(* Logix 5000 project; controller GP1 vendor 1 type 14 code 155 rev 32.11; software revision 32.01; part 2 of 2 *)
(* tags used below, declared in another part *)
   CERRARSESION : BOOL;
   ING_ACCESS : BOOL;
   LOGOUT : BOOL;
   MTTO_ACCESS : BOOL;
   ACT1_OFF : BOOL;   // TROQUEL OFF
   ACT2_OFF : BOOL;   // CORTE SUPERIOR OFF
   ACT3_OFF : BOOL;   // NAVAJA 1 OFF
   ACT5_OFF : BOOL;   // CLAMP OFF
   EVBI0_AUTO_OFF : BOOL;   // NAVAJAS 3 OFF AUTO
   EVBI0_AUTO_ON : BOOL;   // NAVAJAS 3 ON AUTO
   EVBI0_MAN_OFF : BOOL;   // NAVAJAS 3 OFF MANUAL
   EVBI0_MAN_ON : BOOL;   // NAVAJAS 3 ON MANUAL
   EVBI0_OFF : BOOL;   // NAVAJAS 3 OFF
   EVBI0_ON : BOOL;   // NAVAJAS 3 ON
   EVBI1_AUTO_OFF : BOOL;   // TROQUEL OFF AUTO
   EVBI1_AUTO_ON : BOOL;   // TROQUEL ON AUTO
   EVBI1_MAN_OFF : BOOL;   // TROQUEL OFF MANUAL
   EVBI1_MAN_ON : BOOL;   // TROQUEL ON MANUAL
   EVBI1_OFF : BOOL;   // TROQUEL OFF
   EVBI1_ON : BOOL;   // TROQUEL ON
   EVBI2_AUTO_OFF : BOOL;   // CLAMP OFF AUTO
   EVBI2_AUTO_ON : BOOL;   // CLAMP ON AUTO
   EVBI2_MAN_OFF : BOOL;   // CLAMP OFF MANUAL
   EVBI2_MAN_ON : BOOL;   // CLAMP ON MANUAL
   EVBI2_OFF : BOOL;   // CLAMP OFF
   EVBI2_ON : BOOL;   // CLAMP ON
   EVBI3_AUTO_OFF : BOOL;   // NAVAJA 1 OFF AUTO
   EVBI3_AUTO_ON : BOOL;   // NAVAJA 1 ON AUTO
   EVBI3_MAN_OFF : BOOL;   // NAVAJA 1 OFF MANUAL
   EVBI3_MAN_ON : BOOL;   // NAVAJA 1 ON MANUAL
   EVBI3_OFF : BOOL;   // NAVAJA 1 OFF
   EVBI3_ON : BOOL;   // NAVAJA 1 ON
   EVBI4_OFF : BOOL;   // CLAMP VERTICAL OFF
   EVBI4_ON : BOOL;   // CLAMP VERTICAL ON
   EVBI5_AUTO_OFF : BOOL;   // CORTE SUPERIOR OFF AUTO
   EVBI5_AUTO_ON : BOOL;   // CORTE SUPERIOR ON AUTO
   EVBI5_MAN_OFF : BOOL;   // CORTE SUPERIOR OFF MANUAL
   EVBI5_MAN_ON : BOOL;   // CORTE SUPERIOR ON MANUAL
   EVBI5_OFF : BOOL;   // CORTE SUPERIOR OFF
   EVBI5_ON : BOOL;   // CORTE SUPERIOR ON
   EVBI6_OFF : BOOL;   // CLAMP HORIZONTAL OFF
   EVBI6_ON : BOOL;   // CLAMP HORIZONTAL ON
   EVMONO1_AUTO_ON : BOOL;   // TOPE_AUTO_ON
   EVMONO1_MAN_ON : BOOL;
   EVMONO_ON : BOOL;   // TOPE ON
   REARMY_BUTTON : BOOL;
   RESET_COUNTER : BOOL;
   TCLAMP : TIMER;
   USER : DINT;
   WORKING : BOOL;
(* MainProgram, continued *)

ROUTINE OUTPUTS   (* ladder *)
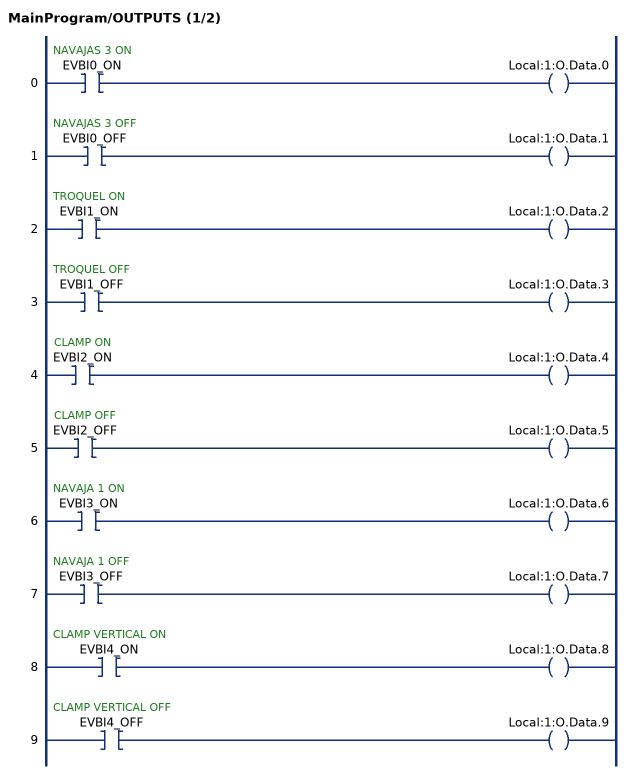
   0: XIC(EVBI0_ON)OTE(Local:1:O.Data.0);
   1: XIC(EVBI0_OFF)OTE(Local:1:O.Data.1);
   2: XIC(EVBI1_ON)OTE(Local:1:O.Data.2);
   3: XIC(EVBI1_OFF)OTE(Local:1:O.Data.3);
   4: XIC(EVBI2_ON)OTE(Local:1:O.Data.4);
   5: XIC(EVBI2_OFF)OTE(Local:1:O.Data.5);
   6: XIC(EVBI3_ON)OTE(Local:1:O.Data.6);
   7: XIC(EVBI3_OFF)OTE(Local:1:O.Data.7);
   8: XIC(EVBI4_ON)OTE(Local:1:O.Data.8);
   9: XIC(EVBI4_OFF)OTE(Local:1:O.Data.9);
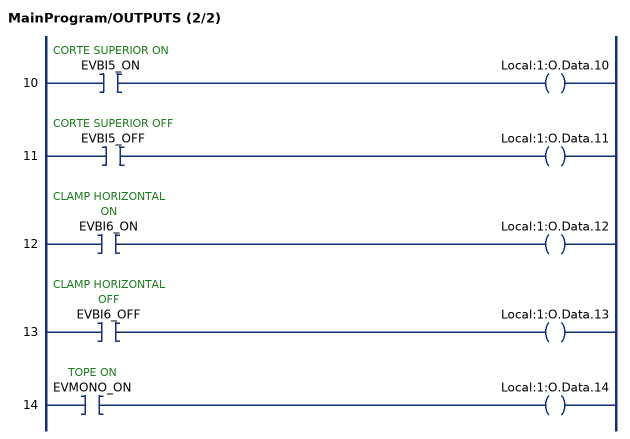
   10: XIC(EVBI5_ON)OTE(Local:1:O.Data.10);
   11: XIC(EVBI5_OFF)OTE(Local:1:O.Data.11);
   12: XIC(EVBI6_ON)OTE(Local:1:O.Data.12);
   13: XIC(EVBI6_OFF)OTE(Local:1:O.Data.13);
   14: XIC(EVMONO_ON)OTE(Local:1:O.Data.14);
END_ROUTINE

ROUTINE USERS   (* ladder *)
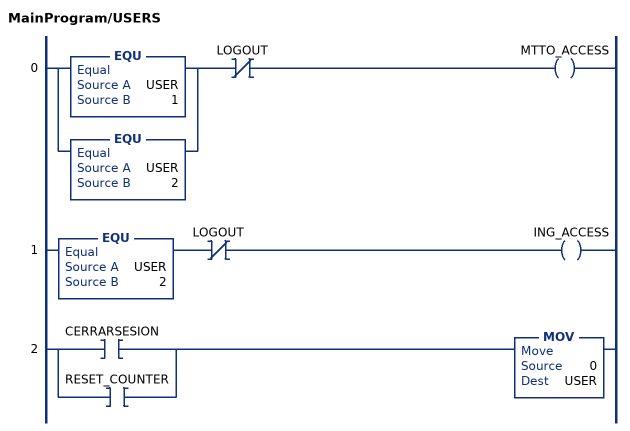
   0: [EQU(USER,1) ,EQU(USER,2) ]XIO(LOGOUT)OTE(MTTO_ACCESS);
   1: EQU(USER,2)XIO(LOGOUT)OTE(ING_ACCESS);
   2: [XIC(CERRARSESION) ,XIC(RESET_COUNTER) ]MOV(0,USER);
END_ROUTINE

ROUTINE VALVES_ACTIV   (* ladder *)
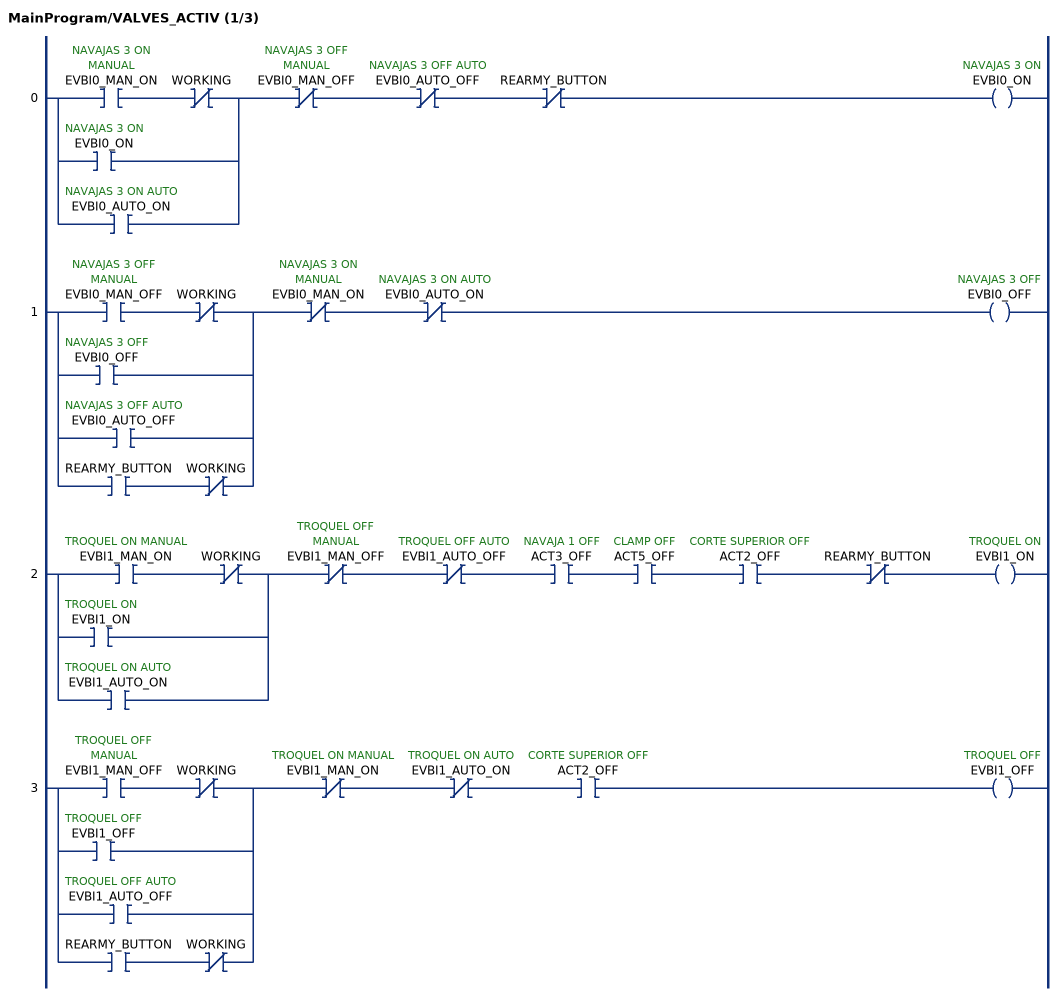
   0: [XIC(EVBI0_MAN_ON) XIO(WORKING) ,XIC(EVBI0_ON) ,XIC(EVBI0_AUTO_ON) ]XIO(EVBI0_MAN_OFF)XIO(EVBI0_AUTO_OFF)XIO(REARMY_BUTTON)OTE(EVBI0_ON);
   1: [XIC(EVBI0_MAN_OFF) XIO(WORKING) ,XIC(EVBI0_OFF) ,XIC(EVBI0_AUTO_OFF) ,XIC(REARMY_BUTTON) XIO(WORKING) ]XIO(EVBI0_MAN_ON)XIO(EVBI0_AUTO_ON)OTE(EVBI0_OFF);
   2: [XIC(EVBI1_MAN_ON) XIO(WORKING) ,XIC(EVBI1_ON) ,XIC(EVBI1_AUTO_ON) ]XIO(EVBI1_MAN_OFF)XIO(EVBI1_AUTO_OFF)XIC(ACT3_OFF)XIC(ACT5_OFF)XIC(ACT2_OFF)XIO(REARMY_BUTTON)OTE(EVBI1_ON);
   3: [XIC(EVBI1_MAN_OFF) XIO(WORKING) ,XIC(EVBI1_OFF) ,XIC(EVBI1_AUTO_OFF) ,XIC(REARMY_BUTTON) XIO(WORKING) ]XIO(EVBI1_MAN_ON)XIO(EVBI1_AUTO_ON)XIC(ACT2_OFF)OTE(EVBI1_OFF);
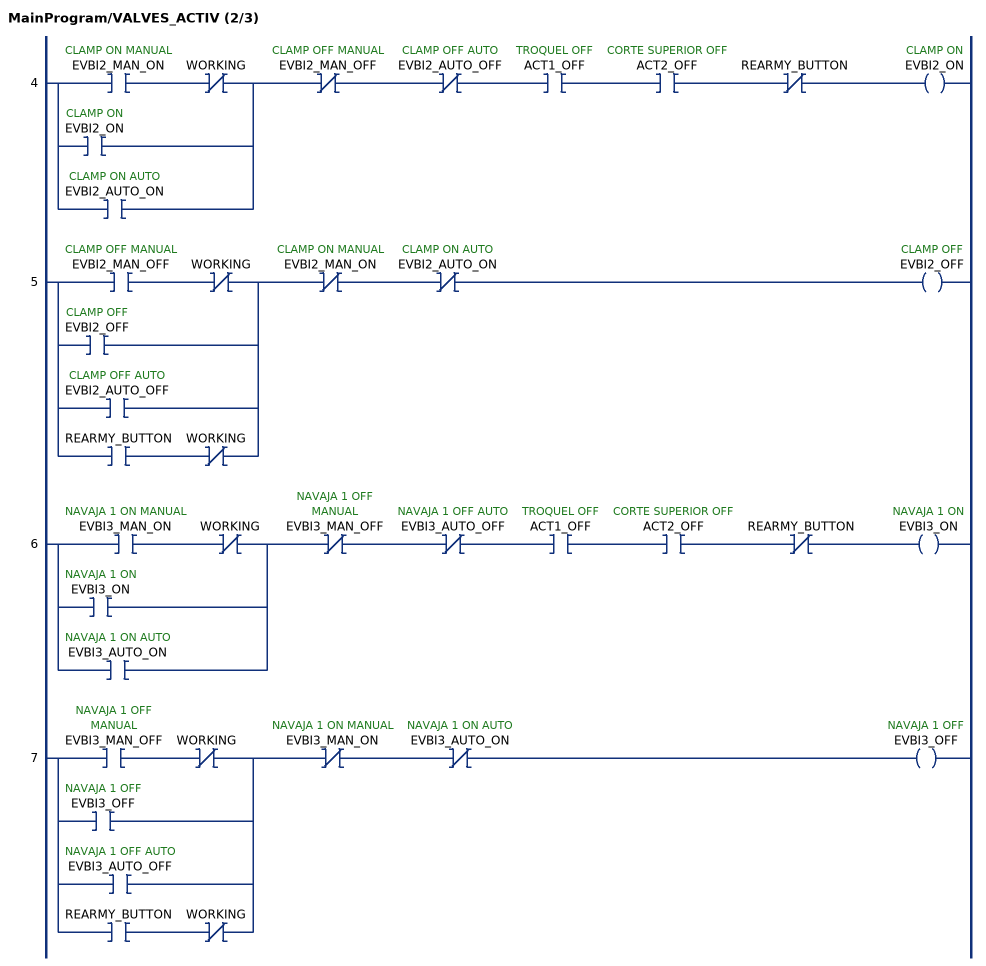
   4: [XIC(EVBI2_MAN_ON) XIO(WORKING) ,XIC(EVBI2_ON) ,XIC(EVBI2_AUTO_ON) ]XIO(EVBI2_MAN_OFF)XIO(EVBI2_AUTO_OFF)XIC(ACT1_OFF)XIC(ACT2_OFF)XIO(REARMY_BUTTON)OTE(EVBI2_ON);
   5: [XIC(EVBI2_MAN_OFF) XIO(WORKING) ,XIC(EVBI2_OFF) ,XIC(EVBI2_AUTO_OFF) ,XIC(REARMY_BUTTON) XIO(WORKING) ]XIO(EVBI2_MAN_ON)XIO(EVBI2_AUTO_ON)OTE(EVBI2_OFF);
   6: [XIC(EVBI3_MAN_ON) XIO(WORKING) ,XIC(EVBI3_ON) ,XIC(EVBI3_AUTO_ON) ]XIO(EVBI3_MAN_OFF)XIO(EVBI3_AUTO_OFF)XIC(ACT1_OFF)XIC(ACT2_OFF)XIO(REARMY_BUTTON)OTE(EVBI3_ON);
   7: [XIC(EVBI3_MAN_OFF) XIO(WORKING) ,XIC(EVBI3_OFF) ,XIC(EVBI3_AUTO_OFF) ,XIC(REARMY_BUTTON) XIO(WORKING) ]XIO(EVBI3_MAN_ON)XIO(EVBI3_AUTO_ON)OTE(EVBI3_OFF);
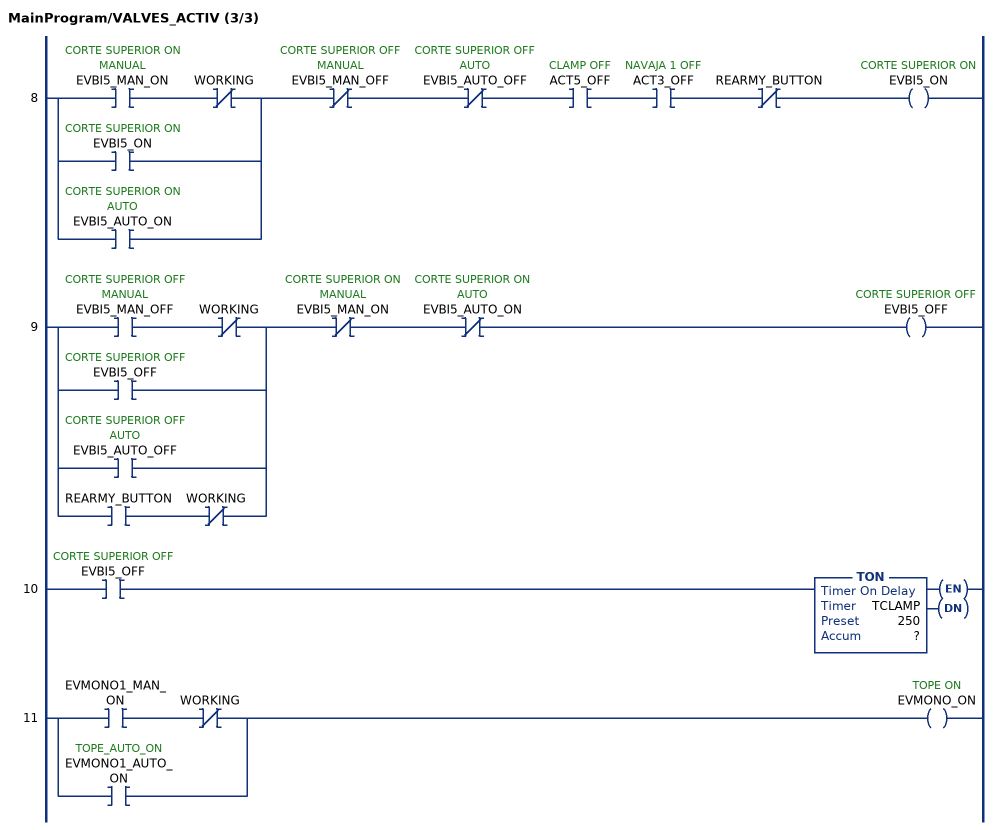
   8: [XIC(EVBI5_MAN_ON) XIO(WORKING) ,XIC(EVBI5_ON) ,XIC(EVBI5_AUTO_ON) ]XIO(EVBI5_MAN_OFF)XIO(EVBI5_AUTO_OFF)XIC(ACT5_OFF)XIC(ACT3_OFF)XIO(REARMY_BUTTON)OTE(EVBI5_ON);
   9: [XIC(EVBI5_MAN_OFF) XIO(WORKING) ,XIC(EVBI5_OFF) ,XIC(EVBI5_AUTO_OFF) ,XIC(REARMY_BUTTON) XIO(WORKING) ]XIO(EVBI5_MAN_ON)XIO(EVBI5_AUTO_ON)OTE(EVBI5_OFF);
   10: XIC(EVBI5_OFF)TON(TCLAMP,?,?);
   11: [XIC(EVMONO1_MAN_ON) XIO(WORKING) ,XIC(EVMONO1_AUTO_ON) ]OTE(EVMONO_ON);
END_ROUTINE
END_PROGRAM
